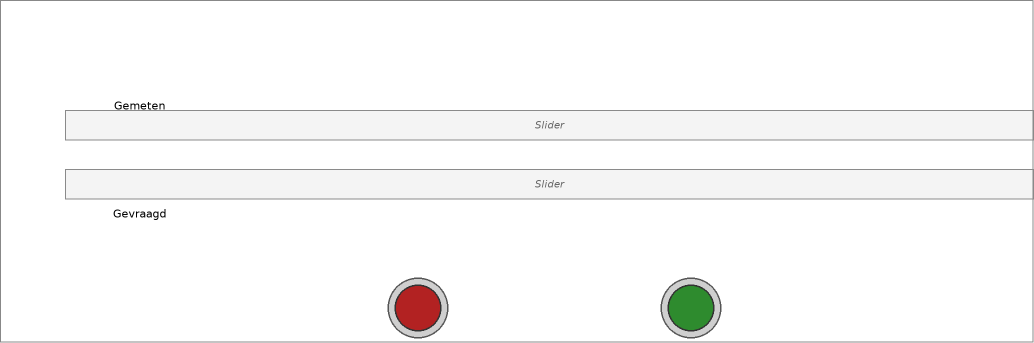
VISUALIZATION Visu  // 1034x343
    Lamp1 (656,273 70x70), variable: MAIN.bGreen, style: Lamp-Lamp1-Green
    Lamp1 (383,273 70x70), variable: MAIN.bRed, style: Lamp-Lamp1-Red
    Slider (65,110 969x30), variable: MAIN.nGemeten, scale 0..32767
    Slider (65,169 969x30), variable: MAIN.nGevraagd, scale 0..15
    Label (65,199 150x30), "Gevraagd"
    Label (65,91 150x30), "Gemeten"
END_VISUALIZATION

(* stored: Version 1.1.0.1, ProductVersion 3.1.4024.12
   Visu Visu: Id {8ab8426a-a07c-4672-a45a-2aaefbf3827f} *)
